Omron Sysmac Studio project distributing_station_tick_tock_17 (Sysmac Studio 1.54.0.64019, StandardProject)

# Controller new_Controller_0: NJ301-1100 version 1.14
Units and slaves: Node1 : NX-ECC201 (E001); Unit 1 : NX-PC0020 (N1); Unit 2 : NX-ID5442 (N2); Unit 3 : NX-PC0010 (N3); Unit 4 : NX-PC0020 (N4); Unit 5 : NX-OD5121 (N5); Unit 6 : NX-PC0010 (N6); Power Supply : NJ-Px3001; CPU : NJ301-1100; 0 [Unit 0] : CJ1W-AD041-V1 (J01); 1 [Unit 1] : CJ1W-DA041 (J02); 2 : CJ1W-ID211 (J03); 3 : CJ1W-OC211 (J04)
Task PrimaryTask (priority 4, period or condition 1000): Program0

VAR_GLOBAL
    Station_1B2 : BOOL;  (* Ejection Cylinder Extended; at IOBus://rack#0/slot#2/Ch1_In/Ch1_In01; published *)
    Station_1B1 : BOOL;  (* Ejection Cylinder retracted; at IOBus://rack#0/slot#2/Ch1_In/Ch1_In02; published *)
    Station_2B1 : BOOL;  (* Workpiece gripped; at IOBus://rack#0/slot#2/Ch1_In/Ch1_In03; published *)
    Station_3S1 : BOOL;  (* arm_in_magazine; at IOBus://rack#0/slot#2/Ch1_In/Ch1_In04; published *)
    Station_3S2 : BOOL;  (* arm_in_downstream; at IOBus://rack#0/slot#2/Ch1_In/Ch1_In05; published *)
    Station_B4 : BOOL;  (* Magzine empty; at IOBus://rack#0/slot#2/Ch1_In/Ch1_In06; published *)
    Panel_S1 : BOOL;  (* start_button; at IOBus://rack#0/slot#2/Ch1_In/Ch1_In08; published *)
    Panel_S2 : BOOL;  (* stop_button; at IOBus://rack#0/slot#2/Ch1_In/Ch1_In09; published *)
    Panel_S4 : BOOL;  (* reset_button; at IOBus://rack#0/slot#2/Ch1_In/Ch1_In11; published *)
    Station_1Y1 : BOOL;  (* Magzine eject; at IOBus://rack#0/slot#3/Ch1_Out/Ch1_Out00; published *)
    Station_2Y1 : BOOL;  (* Vacuum on; at IOBus://rack#0/slot#3/Ch1_Out/Ch1_Out01; published *)
    Station_2Y2 : BOOL;  (* Ejector_Pulse_On; at IOBus://rack#0/slot#3/Ch1_Out/Ch1_Out02; published *)
    Station_3Y1 : BOOL;  (* arm_2_magazine; at IOBus://rack#0/slot#3/Ch1_Out/Ch1_Out03; published *)
    Station_3Y2 : BOOL;  (* arm_2_downstream; at IOBus://rack#0/slot#3/Ch1_Out/Ch1_Out04; published *)
    Station_H1 : BOOL;  (* start light; at IOBus://rack#0/slot#3/Ch1_Out/Ch1_Out08; published *)
    Station_H2 : BOOL;  (* reset light; at IOBus://rack#0/slot#3/Ch1_Out/Ch1_Out09; published *)
    Panel_H3 : BOOL;  (* Q1 light; at IOBus://rack#0/slot#3/Ch1_Out/Ch1_Out10; published *)
    Panel_H4 : BOOL;  (* Q2 light; at IOBus://rack#0/slot#3/Ch1_Out/Ch1_Out11; published *)
END_VAR

PROGRAM Program0
VAR
    FB_Panel_1 : FB_Panel;
    Panel : BOOL;
    run_mode : BOOL;
    stop_mode : BOOL;
    reset_mode : BOOL;
    FB_Actuator_T1_1 : FB_Actuator_T1;
    def : TIME;
    timer_t1 : TON;
END_VAR
VAR_EXTERNAL
    Station_3S1 : BOOL;
    Panel_S2 : BOOL;
    Station_3Y2 : BOOL;
    Station_3S2 : BOOL;
    Panel_S1 : BOOL;
    Station_3Y1 : BOOL;
    Panel_S4 : BOOL;
    Station_H1 : BOOL;
    Station_H2 : BOOL;
    Panel_H4 : BOOL;
    Panel_H3 : BOOL;
END_VAR

(* Section Section0: ladder, written here as Structured Text *)

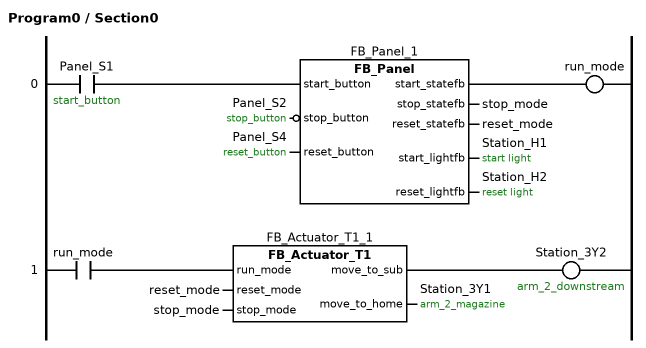
(* Rung 0 *)
FB_Panel_1(start_button := Panel_S1, stop_button := NOT Panel_S2, reset_button := Panel_S4, stop_statefb => stop_mode, reset_statefb => reset_mode, start_lightfb => Station_H1, reset_lightfb => Station_H2);
run_mode := FB_Panel_1.start_statefb;
(* Rung 1 *)
FB_Actuator_T1_1(run_mode := run_mode, reset_mode := reset_mode, stop_mode := stop_mode, move_to_home => Station_3Y1);
Station_3Y2 := FB_Actuator_T1_1.move_to_sub;
END_PROGRAM

FUNCTION_BLOCK FB_Panel
VAR
    flip_flop : RS;
    flip_flop2 : RS;
END_VAR
VAR_OUTPUT
    start_statefb : BOOL;
    stop_statefb : BOOL;
    reset_statefb : BOOL;
END_VAR
VAR_INPUT
    start_button : BOOL := False;
    stop_button : BOOL := False;
    reset_button : BOOL := False;
END_VAR
VAR_OUTPUT
    start_lightfb : BOOL;
    reset_lightfb : BOOL;
END_VAR
(* ladder, written here as Structured Text *)

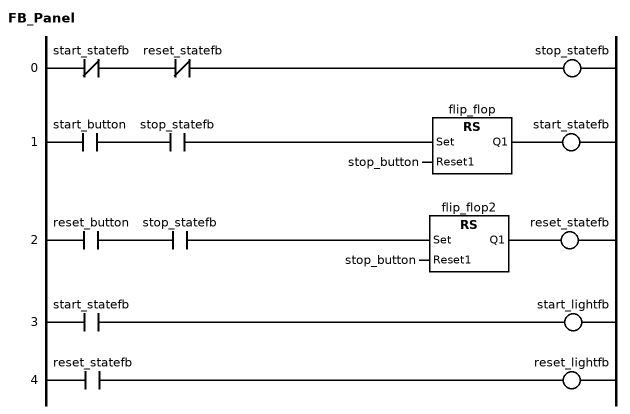
(* Rung 0 *)
stop_statefb := NOT start_statefb AND NOT reset_statefb;
(* Rung 1 *)
flip_flop(Set := start_button AND stop_statefb, Reset1 := stop_button);
start_statefb := flip_flop.Q1;
(* Rung 2 *)
flip_flop2(Set := reset_button AND stop_statefb, Reset1 := stop_button);
reset_statefb := flip_flop2.Q1;
(* Rung 3 *)
start_lightfb := start_statefb;
(* Rung 4 *)
reset_lightfb := reset_statefb;
END_FUNCTION_BLOCK

FUNCTION_BLOCK FB_Actuator_T1
VAR
    flip_flop_1 : RS;
    flip_flop_2 : RS;
    st : BOOL;
    Panel : BOOL;
    move_to_sub_m : BOOL;
    reset_to_home : BOOL;
    timer_t1 : TON;
    flip_flop_3 : RS;
END_VAR
VAR_INPUT
    run_mode : BOOL;
    reset_mode : BOOL;
END_VAR
VAR_OUTPUT
    move_to_sub : BOOL;
    error_mode : BOOL;
    move_to_home : BOOL;
END_VAR
VAR_INPUT
    stop_mode : BOOL;
END_VAR
VAR_EXTERNAL
    Station_3S1 : BOOL;
    Station_3Y1 : BOOL;
    Station_3S2 : BOOL;
    Station_3Y2 : BOOL;
END_VAR
(* ladder, written here as Structured Text *)

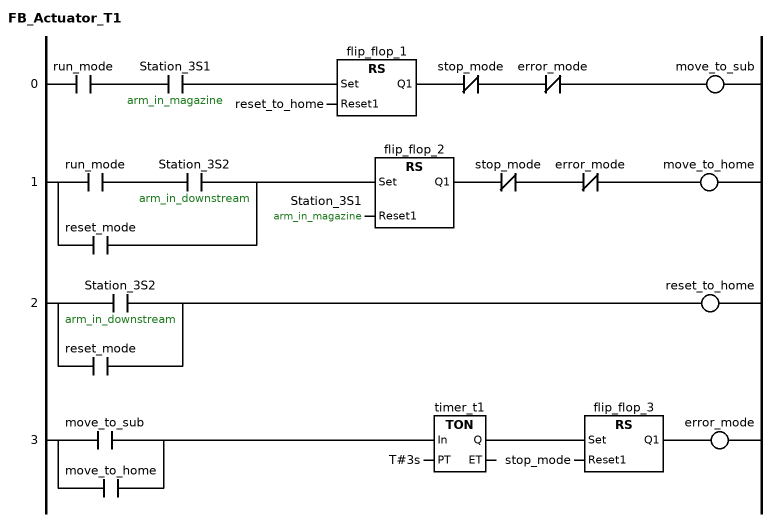
(* Rung 0 *)
flip_flop_1(Set := run_mode AND Station_3S1, Reset1 := reset_to_home);
move_to_sub := flip_flop_1.Q1 AND NOT stop_mode AND NOT error_mode;
(* Rung 1 *)
flip_flop_2(Set := (run_mode AND Station_3S2) OR reset_mode, Reset1 := Station_3S1);
move_to_home := flip_flop_2.Q1 AND NOT stop_mode AND NOT error_mode;
(* Rung 2 *)
reset_to_home := Station_3S2 OR reset_mode;
(* Rung 3 *)
timer_t1(In := move_to_sub OR move_to_home, PT := T#3s);
flip_flop_3(Set := timer_t1.Q, Reset1 := stop_mode);
error_mode := flip_flop_3.Q1;
END_FUNCTION_BLOCK